// TIA Portal V20 export
TYPE "IO_VSD"
   STRUCT
      IN { ExternalAccessible := 'False'; ExternalVisible := 'False'; ExternalWritable := 'False'} : Struct
         Trip : Bool;
         FwdFb : Bool;
         RevFb : Bool;
         SpeedFb : Real;
      END_STRUCT;
      OUT { ExternalAccessible := 'False'; ExternalVisible := 'False'; ExternalWritable := 'False'} : Struct
         FwdCmd : Bool;
         RevCmd : Bool;
         SpeedCmd : Real;
      END_STRUCT;
   END_STRUCT;
END_TYPE
